FUNCTION_BLOCK F_SEL_E_4 (* selection event-based selection) (generic FB) *)
  (* Standard: 61131-3; Classification: standard selection function; Description: Copyright (c) 2012, 2022 TU Wien ACIN, HR Agrartechnik GmbH This program and the accompanying materials are made available under the terms of the Eclipse Public License 2.0 which is available at https://www.eclipse.org/legal/epl-2.0/ SPDX-License-Identifier: EPL-2.0 *)
  (* Version 3.0, 2025-04-14, Patrick Aigner, changed package *)
  (* Version 1.1, 2022-08-04, Franz Höpfinger, HR Agrartechnik GmbH *)
  (* Version 1.0, 2012-03-25, Monika Wenger, TU Wien ACIN *)
  PACKAGE eclipse4diac::utils::selection;
  {SET_ATTRIBUTE(eclipse4diac::core::GenericClassName, 'GEN_F_SEL_E')}
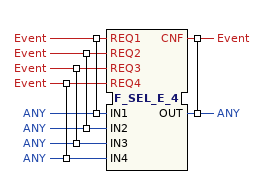
  EVENT_INPUT
    REQ1 WITH IN1;
    REQ2 WITH IN2;
    REQ3 WITH IN3;
    REQ4 WITH IN4;
  END_EVENT
  EVENT_OUTPUT
    CNF WITH OUT; (* Confirmation of Requested Service *)
  END_EVENT
  VAR_INPUT
    IN1 : ANY; (* Selectable input variable *)
    IN2 : ANY; (* Selectable input variable *)
    IN3 : ANY; (* Selectable input variable *)
    IN4 : ANY; (* Selectable input variable *)
  END_VAR
  VAR_OUTPUT
    OUT : ANY; (* Selected input *)
  END_VAR
END_FUNCTION_BLOCK
